TYPE ST_IOInputSimul :
STRUCT
	IxAru :BOOL;
END_STRUCT
END_TYPE

(* stored: Version 1.1.0.1, ProductVersion 3.1.4020.6
   DUT ST_IOInputSimul: Id {65db8fb7-7793-4d51-ac3e-b549fd087b69} *)
